{attribute 'GeneratedUsingTerminal: KL3361-0003'}
{attribute addProperty BoxType "KL3361-0003"}
{attribute addProperty Id "Channel_1AT %Q*Channel_78571FB40"}
{attribute addProperty CRC "1942717114"}
{attribute addProperty Size "0"}
TYPE KL_73CB82BA :
STRUCT
	{attribute addProperty Name "Channel_1"}
	Channel_1 : Channel_78571FB4;
END_STRUCT
END_TYPE

(* stored: Version 1.2.0.0, ProductVersion 3.1.4024.9
   DUT KL_73CB82BA: Id {550c9fa1-f40f-45ff-ae2d-968cd8319079} *)
